FUNCTION_BLOCK FB_MotorWrapper IMPLEMENTS IF_Actuator
VAR_INPUT
END_VAR
VAR_OUTPUT
END_VAR
VAR_IN_OUT
	Axis : AXIS_REF;
END_VAR

VAR
	// MC2 Motion Function Blocks
    fbPower       : MC_Power;
    fbReset       : MC_Reset;
	fbReadStatus  : MC_ReadStatus;
    fbMoveAbs     : MC_MoveAbsolute;
    fbMoveRel     : MC_MoveRelative;
	fbMoveVel	  : MC_MoveVelocity;
	fbSetPos	  : MC_SetPosition;
    fbHome        : MC_Home;
	fbReadPos	  : MC_ReadActualPosition;
    fbStop        : MC_Stop;
	fbHalt		  : MC_Halt;
	fbJog		  : MC_Jog;
    rTrigStop     : R_TRIG;

    fSetPosAbs    : LREAL;
    fSetPosRel    : LREAL;
    bAbsRequest   : BOOL;
    bRelRequest   : BOOL;
    bPowerRequest : BOOL;
    bResetRequest : BOOL;
    bDisableReq   : BOOL;
	
	//Stop()
    bStopExecute     : BOOL;
    bStopRequested   : BOOL;
	bStopDone		 : BOOL;
	
	//GetStatus()
    stStatus       	 : ST_ActuatorStatus;
	stReadStatus	 : ST_AxisReadStatus;
	lastPosition 	 : LREAL := 0.0;
	deltaPos 		 : LREAL;
    bDetectedMovement: BOOL  := FALSE;
    debugSensorValue : BOOL;
	
	//Home()
	bStartDelay		 : BOOL := FALSE;
	tonHoming 		 : TON;
	bhomeExecute	 : BOOL := FALSE;
	bHomeRequest 	 : BOOL := FALSE;

	bExecuteMove	 : BOOL;
	bHomeSensorValue : BOOL;
	bHomeInProgress  : BOOL := FALSE;
	bStartMoveVel	 : BOOL;
	bWaitingForSensorOff : BOOL;
	bWaitingForStop	: BOOL;
	bStartHoming	: BOOL;
	
	//ReadStatus()
	bReadStatusExecute 	: BOOL;
    bReadStatusRequested: BOOL;
	
	//MoveAbs()
	bMoveAbsExecute 	: BOOL;
    bMoveAbsRequested 	: BOOL;
	bMoveAbsDone		: BOOL;
	bMoveAbsStarted		: BOOL;
	rtMoveAbsDone 		: R_TRIG; 
    tonMoveAbs    		: TON;    
    tMoveAbsTout  		: TIME := T#60S;
	tonAbsInWin         : TON;         // estabilidade da janela de posição
	rAbsPosTol          : LREAL := 0.001; // tolerância (ajuste ao teu unit)
	tAbsStable          : TIME  := T#100MS; // estabilidade da janela
	tonAbsTimeout       : TON;         // timeout opcional
	tAbsTimeout         : TIME  := T#60S;   // ajuste conforme curso do eixo
	fbReadVel        	: MC_ReadActualVelocity; // se ainda não existir no FB
	tonVelStill      	: TON;                   // estabilidade de "velocidade ~ 0"
	vTolStill        	: LREAL := 0.0001;       // tolerância de velocidade
	rVelAbs          	: LREAL;                 // auxiliar
	rActPrev         	: LREAL;                 // opcional, se preferir medir Δpos
	
	
	//MoveRel()
	bMoveRelExecute 	: BOOL;
    bMoveRelRequested 	: BOOL;
	bMoveRelDone		: BOOL;
	
	//MoveValve()
	rTargetAngle		: LREAL;
	bMoveValveExecute 	: BOOL;
    bMoveValveRequested : BOOL;
	
	//MoveVel()
	bMoveVelExecute 	: BOOL;
    bMoveVelRequested 	: BOOL;
	bMoveVelDone		: BOOL;
	
	//Reset()
	bResetExecute 		: BOOL;
    bResetRequested 	: BOOL;
	bResetDone			: BOOL;
	
	//SetPosition()
	bSetPosExecute 		: BOOL;
    bSetPosRequested	: BOOL;
	bSetPosDone			: BOOL;
	
	
END_VAR

METHOD Disable : BOOL
VAR_INPUT
END_VAR
// Disable (Remove power from axis)
fbPower(Axis := Axis, Enable := FALSE);
stStatus.bEnabled := FALSE;
stStatus.eState := E_ActuatorState.eDisabled;
Disable := TRUE;
END_METHOD

METHOD Enable : BOOL
VAR_INPUT
END_VAR
// Call MC_Power to enable axis
fbPower(Axis := Axis, Enable := TRUE, Enable_Positive := TRUE, Enable_Negative := TRUE);
stStatus.bEnabled := fbPower.Status;
stStatus.bError := fbPower.Error;
stStatus.iErrorCode := fbPower.ErrorID;
IF fbPower.Error THEN
	stStatus.eState := E_ActuatorState.eError;
	stStatus.sMessage := 'Error in PowerUp';
ELSE
	stStatus.eState := E_ActuatorState.eActive;
END_IF;

Enable := fbPower.Status;
END_METHOD

METHOD GetPosition : LREAL
VAR_INPUT
END_VAR
//Get Actual Position of the motor
//fbReadPos(Axis := Axis, Enable := TRUE);
GetPosition := Axis.NcToPlc.ActPos;
END_METHOD

METHOD GetStatus : ST_ActuatorStatus
VAR_INPUT
END_VAR
// Get unified status struct with all feedback for HMI/diagnostics
fbReadPos(Axis := Axis, Enable := TRUE);
stStatus.fPosition := fbReadPos.Position;
stStatus.bBusy := fbMoveAbs.Busy OR fbMoveRel.Busy OR fbHome.Busy OR fbMoveVel.Busy OR bDetectedMovement;
stStatus.bDone := fbMoveAbs.Done OR fbMoveRel.Done OR fbHome.Done;
stStatus.bError := Axis.Status.Error;

// Calc the position diference
deltaPos := fbReadPos.Position - lastPosition;

IF ABS(deltaPos) > 0.1 THEN
    // Detects forward movement
    IF deltaPos > 0 THEN
		stStatus.bMovingFwd := TRUE;
		stStatus.bMovingBck := FALSE;
		bDetectedMovement   := TRUE;
    // Detects backward movement
    ELSIF deltaPos < 0 THEN
        stStatus.bMovingFwd := FALSE;
        stStatus.bMovingBck := TRUE;
		bDetectedMovement   := TRUE;
    END_IF
ELSE
    // No movement
    stStatus.bMovingFwd := FALSE;
    stStatus.bMovingBck := FALSE;
	bDetectedMovement   := FALSE;
END_IF

lastPosition := fbReadPos.Position;

// Prioritize error messages by source
IF stStatus.bError THEN
	stStatus.eState := E_ActuatorState.eError;
	IF fbPower.Error THEN
		stStatus.sMessage := 'Error in PowerUp';
	ELSIF fbMoveAbs.Error THEN
		stStatus.sMessage := 'Error in MoveAbsolute';
	ELSIF fbMoveRel.Error THEN
		stStatus.sMessage := 'Error in MoveRelative';
	ELSIF fbMoveVel.Error THEN
		stStatus.sMessage := 'Error in MoveVelocity';
	ELSIF fbHome.Error THEN
		stStatus.sMessage := 'Error in Home';
	END_IF
END_IF;

//return
GetStatus := stStatus;
END_METHOD

METHOD Home : BOOL
VAR_INPUT
	pHomeSensor : POINTER TO BOOL; // home sensor pointer
	rVelocity : LREAL;
    rAcc      : LREAL;
    rDec      : LREAL;
	
END_VAR
VAR
	 rTrigHome : R_TRIG;
	 rTrigMove : R_TRIG;
	 rTrigStop : R_TRIG;
END_VAR
bHomeSensorValue  := pHomeSensor^;
IF NOT bHomeRequest THEN
	Home := FALSE;
	bHomeRequest := TRUE;
END_IF

//IF NOT GVL_Motion.bInitialHomingDone THEN
	
	IF bHomeRequest AND NOT bHomeInProgress AND bHomeSensorValue THEN
		bExecuteMove 	:= TRUE;
		bHomeInProgress := TRUE;
	END_IF
	
	IF bHomeRequest AND NOT bHomeInProgress THEN
		bExecuteMove 	:= FALSE;
	
		// If the sensor is already active, skip movement and go to homing directly
		IF NOT bHomeSensorValue THEN
			bStartDelay := TRUE;
			bHomeInProgress := TRUE;
		ELSE
			bExecuteMove := TRUE;
			bHomeInProgress := TRUE;
		END_IF
	END_IF
	
	fbMoveVel(Axis := Axis, Execute := bExecuteMove, Velocity := rVelocity, Acceleration := rAcc, Deceleration := rDec, direction := 1); 
	
	fbStop(Axis := Axis, Execute := bStopExecute, Deceleration := 100);
	
	IF bHomeSensorValue THEN
		//fbMoveVel(Axis := Axis, Execute := bExecuteMove, Velocity := rVelocity, Acceleration := rAcc, Deceleration := rDec, direction := 1); //15, 20, 20
		stStatus.sMessage := 'Seeking home sensor...';
		bStopExecute := FALSE;
	ELSIF NOT bStartDelay THEN
		bExecuteMove := FALSE;
		bStopExecute := TRUE;
		//fbStop(Axis := Axis, Execute := bStopExecute, Deceleration := 10);
	END_IF
	
	IF fbStop.Done THEN
		bStopExecute := FALSE;
		bStartDelay := TRUE;
	END_IF
	
	IF NOT fbStop.Busy THEN
		tonHoming(IN := bStartDelay, PT := T#2S);
	END_IF
	
	IF tonHoming.Q THEN
		bhomeExecute := TRUE;
		stStatus.sMessage := 'Executing MC_Home...';
	END_IF
	
	fbHome(Axis := Axis, Execute := bhomeExecute, Position := 0.0, HomingMode := MC_Direct);
	
	IF fbHome.Done THEN
		stStatus.eState := E_ActuatorState.eIdle;
		stStatus.bError := FALSE;
		stStatus.bDone := TRUE;
		stStatus.sMessage := 'Homing completed';
		bStartDelay  := FALSE;
		bhomeExecute := FALSE;
		tonHoming.IN := FALSE;
		bHomeInProgress := FALSE;
		//GVL_Motion.bMotorsHomeDone := TRUE;
		bHomeRequest := FALSE;
		Home := TRUE;
		RETURN;
	ELSIF fbHome.Error THEN
		stStatus.eState := E_ActuatorState.eError;
		stStatus.bError := TRUE;
		stStatus.iErrorCode := fbHome.ErrorID;
		stStatus.sMessage := 'Error in Homing';
		bhomeExecute := FALSE;
		bStartDelay  := FALSE;
		tonHoming.IN := FALSE;
		bHomeInProgress := FALSE;
		bHomeRequest := FALSE;
		Home := FALSE;
	ELSE
		Home := FALSE;
	END_IF
(*ELSE
	
	IF fbMoveAbs.Done THEN 
		bHomeinProgress := FALSE;
		Home := TRUE;
	END_IF
	
	rTrigMove(CLK := bHomeRequest AND NOT bHomeInProgress);
	
	// If homing previously done then Move to zero position
	fbMoveAbs(Axis := Axis, Execute := rTrigMove.Q, Position := 0, velocity := 15, Acceleration := 15, Deceleration := 15);
	bHomeinProgress := TRUE;
	

	
END_IF*)
END_METHOD

METHOD Jog : BOOL
VAR_INPUT
	bFwd : BOOL;
	bBwd : BOOL;
	//rVelocity : LREAL;
END_VAR
// Call the internal motion block
fbJog(
    Axis := Axis,
    JogForward := bFwd,
    JogBackwards := bBwd,
    Mode := MC_JOGMODE_STANDARD_FAST,
);

// Update actuator status
stStatus.bBusy := fbJog.Busy;
stStatus.bDone := fbJog.Done;
stStatus.bError := fbJog.Error;
stStatus.iErrorCode := fbJog.ErrorID;

Jog := fbJog.Busy;
END_METHOD

METHOD MoveAbsolute : BOOL
VAR_INPUT
	rPosition : LREAL;
    rVelocity : LREAL := 10.0;
    rAcc      : LREAL := 20.0;
    rDec      : LREAL := 20.0;
END_VAR
VAR
	rAct : LREAL;
    rErr : LREAL;
    bInWin : BOOL;
    bStandStill : BOOL;
	opts : ST_MoveOptions;
END_VAR
//Standard Output
MoveAbsolute := FALSE;

// Trigger the command request
IF NOT bMoveAbsRequested THEN
    bMoveAbsExecute := TRUE;
    bMoveAbsRequested := TRUE;
END_IF

// MC_MoveAbsolute function block call
opts.IgnorePositionMonitoring := TRUE;   // Standard practice for move commands

fbMoveAbs(
    Axis := Axis,
    Position := rPosition,
    Execute := bMoveAbsExecute, // Execute flag is controlled by the logic below
    Velocity := rVelocity,
    Acceleration := rAcc,
    Deceleration := rDec,
	options := opts
);

// Release the Execute signal once the block gets in busy or error mode
IF fbMoveAbs.Busy OR fbMoveAbs.Error OR fbMoveAbs.CommandAborted THEN
    bMoveAbsExecute := FALSE;
END_IF

// Flag that movement has successfully started
IF fbMoveAbs.Busy THEN
    bMoveAbsStarted := TRUE;
END_IF

// Status mapping to the wrapper's public status structure
stStatus.bBusy := fbMoveAbs.Busy;
stStatus.bDone := fbMoveAbs.Done;
stStatus.bError := fbMoveAbs.Error;
stStatus.iErrorCode := fbMoveAbs.ErrorID;

//Check if there was any erros on the fbMoveAbs block and resets the trigger
IF bMoveAbsRequested AND bMoveAbsStarted AND 
   	NOT fbMoveAbs.Busy AND NOT fbMoveAbs.Done AND NOT fbMoveAbs.Error THEN
		bMoveAbsRequested := FALSE;
    	bMoveAbsStarted := FALSE;
	
		stStatus.bError := TRUE;
		stStatus.iErrorCode := 9001; // Custom code for 'Motion Aborted/Stuck'
		stStatus.sMessage := 'Movement started but was silently aborted (check external Stop/Power).';
END_IF
	
// Finalization — true Done confirmation
IF bMoveAbsRequested AND fbMoveAbs.Done AND bMoveAbsStarted THEN
    bMoveAbsRequested := FALSE;
	bMoveAbsStarted := FALSE;
    MoveAbsolute := TRUE;
    RETURN;
END_IF

// Abort/error handling
IF fbMoveAbs.CommandAborted THEN
    stStatus.eState := E_ActuatorState.eError;
    stStatus.sMessage := 'Command aborted';
END_IF
IF fbMoveAbs.Error THEN
    stStatus.eState := E_ActuatorState.eError;
    stStatus.sMessage := 'Error in Move Motor';
END_IF
END_METHOD

METHOD MoveRelative : BOOL
VAR_INPUT
	Distance : LREAL;
    Velocity : LREAL := 10.0;
    Acc      : LREAL := 20.0;
    Dec      : LREAL := 20.0;
END_VAR
VAR
END_VAR
// Reuse the same logic from MoveAbsolute
IF NOT bMoveRelRequested THEN
    bMoveRelExecute := TRUE;
    bMoveRelRequested := TRUE;
END_IF

IF fbMoveRel.Busy THEN
    bMoveRelExecute := FALSE;
END_IF

// Call the internal motion block
fbMoveRel(
    Axis := Axis,
    Distance := Distance,
    Execute := bMoveRelExecute,
    Velocity := Velocity,
    Acceleration := Acc,
    Deceleration := Dec
);

// Update actuator status
stStatus.bBusy := fbMoveRel.Busy;
stStatus.bDone := fbMoveRel.Done;
stStatus.bError := fbMoveRel.Error;
stStatus.iErrorCode := fbMoveRel.ErrorID;

IF fbMoveRel.Error THEN
    stStatus.eState := E_ActuatorState.eError;
    stStatus.sMessage := 'Error in Move Motor';
END_IF

IF bMoveRelRequested AND NOT fbMoveRel.Busy AND NOT fbMoveRel.Error THEN
    bMoveRelRequested := FALSE;
    MoveRelative := TRUE;
    RETURN;
ELSE
    MoveRelative := FALSE;
END_IF
END_METHOD

METHOD MoveValve : BOOL
VAR_INPUT
	iPosition : USINT;
	rVelocity : LREAL;
	rAcc	  : LREAL;
	rDec	  : LREAL;
END_VAR
// Map logical valve position to angular position
CASE iPosition OF
    1: rTargetAngle := 0.0;
    2: rTargetAngle := 1200.0;
    3: rTargetAngle := 2400.0;
    4: rTargetAngle := 3600.0;
    5: rTargetAngle := 4800.0;
    6: rTargetAngle := 6000.0;
ELSE
    rTargetAngle := 0;
END_CASE

// Reuse the same logic from MoveAbsolute
IF NOT bMoveValveRequested THEN
    bMoveValveExecute := TRUE;
    bMoveValveRequested := TRUE;
END_IF


// Call the internal motion block
fbMoveAbs(
    Axis := Axis,
    Position := rTargetAngle,
    Execute := bMoveValveExecute,
    Velocity := rVelocity,
    Acceleration := rAcc,
    Deceleration := rDec
);

// Update actuator status
stStatus.bBusy := fbMoveAbs.Busy;
stStatus.bDone := fbMoveAbs.Done;
stStatus.bError := fbMoveAbs.Error;
stStatus.iErrorCode := fbMoveAbs.ErrorID;

IF fbMoveAbs.Busy THEN
    bMoveValveExecute := FALSE;
END_IF

IF fbMoveAbs.Error THEN
    stStatus.eState := E_ActuatorState.eError;
    stStatus.sMessage := 'Error in MoveValve';
END_IF

IF bMoveValveRequested AND NOT fbMoveAbs.Busy AND NOT fbMoveAbs.Error THEN
    bMoveValveRequested := FALSE;
    MoveValve := TRUE;
    RETURN;
ELSE
    MoveValve := FALSE;
END_IF
END_METHOD

METHOD MoveVelocity : BOOL
VAR_INPUT
    rVelocity  : LREAL := 10.0;
    rAcc       : LREAL := 20.0;
    rDec       : LREAL := 20.0;
	iDirection : E_PumpDirection;
END_VAR

VAR
	mcDirection: MC_Direction;
END_VAR
// Reuse the same logic from MoveAbsolute
IF NOT bMoveVelRequested THEN
    bMoveVelExecute := TRUE;
    bMoveVelRequested := TRUE;
END_IF

// Get the corect direction
IF iDirection = E_PumpDirection.Forward THEN
	mcDirection := MC_Direction.MC_Positive_Direction;
	ELSE IF iDirection = E_PumpDirection.Backward THEN
		mcDirection := MC_Direction.MC_Negative_Direction;
	ELSE
		mcDirection := MC_Direction.MC_Current_Direction;
	END_IF
END_IF

// Call the internal motion block
fbMoveVel( 	Axis := Axis,
			Execute := bMoveVelExecute,
			Velocity := rVelocity,
			Direction := mcDirection,
			Acceleration := rAcc,
			Deceleration := rDec
);
			
// Update actuator status
stStatus.bBusy := fbMoveVel.Busy;
stStatus.bError := fbMoveVel.Error;
stStatus.iErrorCode := fbMoveVel.ErrorID;

IF fbMoveVel.Busy THEN
    bMoveVelExecute := FALSE;
END_IF

IF fbMoveVel.Error THEN
    stStatus.eState := E_ActuatorState.eError;
    stStatus.sMessage := 'Error in Move Motor';
END_IF

IF bMoveVelRequested AND NOT fbMoveVel.Busy AND NOT fbMoveVel.Error THEN
    bMoveVelRequested := FALSE;
    MoveVelocity := TRUE;
    RETURN;
ELSE
    MoveVelocity := FALSE;
END_IF
END_METHOD

METHOD ReadStatus : ST_AxisReadStatus
VAR_INPUT
END_VAR
//Method to read status by MC_ReadStatus
Axis.ReadStatus();

//Filling up stReadStatus
stReadStatus.Disabled :=  Axis.Status.Disabled;
stReadStatus.Error := Axis.Status.Error;
stReadStatus.ErrorID := Axis.Status.ErrorID;
stReadStatus.Homed := Axis.Status.Homed;
stReadStatus.Operational := Axis.Status.Operational;
stReadStatus.StandStill := Axis.Status.StandStill;

//Return
ReadStatus := stReadStatus;
END_METHOD

METHOD ReadValveStatus : BOOL
VAR_INPUT
END_VAR
Axis.ReadStatus();

IF Axis.Status.Error AND Axis.Status.ErrorID = 16#00004466 THEN
    ReadValveStatus := FALSE;
ELSE
    ReadValveStatus := NOT Axis.Status.Error AND NOT Axis.Status.Disabled;
END_IF
END_METHOD

METHOD Reset : BOOL
VAR_INPUT
END_VAR
VAR
    (* Local helper to clear flags only on very first call of this reset cycle *)
    bFirstCall : BOOL := FALSE;
	stAxisStat : ST_AxisReadStatus;
END_VAR
// ============================================================================
// 0) Default
// ============================================================================
Reset := FALSE;

// Allways read the actual axis state
Axis.ReadStatus();
stAxisStat.Disabled   			:= Axis.Status.Disabled;
stAxisStat.Error      			:= Axis.Status.Error;
stAxisStat.ErrorID    			:= Axis.Status.ErrorID;
stAxisStat.Homed      			:= Axis.Status.Homed;
stAxisStat.Operational			:= Axis.Status.Operational;
stAxisStat.StandStill 			:= Axis.Status.StandStill;
stAxisStat.MotionCommandsLocked	:= Axis.Status.MotionCommandsLocked;

// 0.1) If the axis is NOT in error, there is nothing to reset.
IF NOT stAxisStat.Error AND NOT stAxisStat.MotionCommandsLocked THEN
    // It guarantees a "clean" status.
    stStatus.bError      := FALSE;
    stStatus.iErrorCode  := 0;
    stStatus.sMessage    := '';
    stStatus.eState      := E_ActuatorState.eIdle;

    // Clear internal reset flags
    bResetRequested      := FALSE;
    bResetExecute        := FALSE;
    bResetDone           := FALSE;

    Reset := TRUE;
    RETURN;
END_IF

// ============================================================================
// 1) Detect new Reset() cycle
// 		- Only enters this section when there is actually an error on the axis
// ============================================================================
IF NOT bResetRequested AND NOT bResetExecute AND NOT bResetDone THEN
    bFirstCall     := TRUE;
    bResetRequested:= TRUE;
END_IF

IF bFirstCall THEN
    // --------------------------------------------------------
    // 1.1) Clears all MC's Executes and internal flags.
    // --------------------------------------------------------
    fbPower(Axis := Axis, Enable := FALSE, Enable_Positive := FALSE, Enable_Negative := FALSE);
    fbMoveAbs(Axis := Axis, Execute := FALSE);
    fbMoveRel(Axis := Axis, Execute := FALSE);
    fbMoveVel(Axis := Axis, Execute := FALSE);
    fbHome(Axis := Axis, Execute := FALSE);
    fbSetPos(Axis := Axis, Execute := FALSE);
    fbStop(Axis := Axis, Execute := FALSE);
    fbHalt(Axis := Axis, Execute := FALSE);
    fbReadStatus(Axis := Axis, Enable := FALSE);
    fbReadPos(Axis := Axis, Enable := FALSE);
	fbReset(Axis := Axis, Execute := FALSE);

    bPowerRequest         := FALSE;
    bDisableReq           := FALSE;

    bAbsRequest           := FALSE;
    bRelRequest           := FALSE;

    bReadStatusRequested  := FALSE;
    bReadStatusExecute    := FALSE;

    // Move Abs
    bMoveAbsRequested     := FALSE;
    bMoveAbsExecute       := FALSE;
    bMoveAbsDone          := FALSE;
    bMoveAbsStarted       := FALSE;

    // Move Rel
    bMoveRelRequested     := FALSE;
    bMoveRelExecute       := FALSE;
    bMoveRelDone          := FALSE;

    // Move Valve
    bMoveValveRequested   := FALSE;
    bMoveValveExecute     := FALSE;

    // Move Vel
    bMoveVelRequested     := FALSE;
    bMoveVelExecute       := FALSE;
    bMoveVelDone          := FALSE;

    // SetPos
    bSetPosRequested      := FALSE;
    bSetPosExecute        := FALSE;
    bSetPosDone           := FALSE;

    // Stop / Halt / Home
    bStopRequested        := FALSE;
    bStopExecute          := FALSE;
    bStopDone             := FALSE;
    bHomeRequest          := FALSE;
    bHomeInProgress       := FALSE;
    bStartHoming          := FALSE;
    bStartMoveVel         := FALSE;
    bWaitingForSensorOff  := FALSE;
    bWaitingForStop       := FALSE;

    // Flags do reset
    bResetRequest         := FALSE;
    bResetRequested       := TRUE;
    bResetDone            := FALSE;

    tonMoveAbs(IN := FALSE);
    tonAbsInWin(IN := FALSE);
    tonHoming(IN := FALSE);
    tonVelStill(IN := FALSE);
    tonAbsTimeout(IN := FALSE);

    rtMoveAbsDone(CLK := FALSE);
    rTrigStop(CLK := FALSE);

    stStatus.bBusy        := FALSE;
    stStatus.bError       := TRUE;             // still error
    stStatus.iErrorCode   := stAxisStat.ErrorID;
    stStatus.sMessage     := 'Resetting axis error...';
    stStatus.eState       := E_ActuatorState.eError;

    bFirstCall := FALSE;
END_IF

// ============================================================================
// 2) Triggers MC_Reset 1x per reset cycle
// ============================================================================
IF bResetRequested AND NOT bResetExecute AND NOT bResetDone THEN
    bResetExecute := TRUE;
END_IF

fbReset(
    Axis    := Axis,
    Execute := bResetExecute
);

// ============================================================================
// 3) MC_Reset error handling
// ============================================================================
IF fbReset.Error THEN
    stStatus.bError      := TRUE;
    stStatus.iErrorCode  := fbReset.ErrorID;
    stStatus.sMessage    := 'Error in MC_Reset';
    stStatus.eState      := E_ActuatorState.eError;

    bResetExecute        := FALSE;
    bResetRequested      := FALSE;
    bResetDone           := FALSE;

    Reset := FALSE;
    RETURN;
END_IF

// MC_Reset's Done
IF fbReset.Done THEN
    bResetExecute := FALSE;
    bResetDone    := TRUE;
END_IF

// ============================================================================
// 4) Finalization: only concludes if the axis really recovered from the error.
// ============================================================================
IF bResetDone AND NOT fbReset.Busy THEN
    // reads the axis status again
    Axis.ReadStatus();
    IF NOT Axis.Status.Error AND NOT Axis.Status.MotionCommandsLocked THEN
        // Success
        stStatus.bError      := FALSE;
        stStatus.iErrorCode  := 0;
        stStatus.sMessage    := '';
        stStatus.eState      := E_ActuatorState.eIdle;

        bResetRequested      := FALSE;
        bResetDone           := FALSE;

        Reset := TRUE;
        RETURN;
    ELSE
        // Still in error (e.g., 0x4650, 0x4260, etc.)
		// Starts another MC_Reset cycle
        bResetDone     := FALSE;
        bResetExecute  := TRUE;
        // Reset remains FALSE until the error is actually cleared.
    END_IF
END_IF


(* Old Reset procedure before 2025's Nov27th
// ============================================================================
// 0) Default return
// ============================================================================
Reset := FALSE;

// ============================================================================
// 1) First call of Reset() in this cycle: clear ALL internal flags and MC executes
// ============================================================================

// If neither a reset request nor a reset execution is active, this is a NEW reset cycle
IF NOT bResetRequested AND NOT bResetExecute AND NOT bResetDone THEN
    bFirstCall := TRUE;
    bResetRequested := TRUE;
END_IF

IF bFirstCall THEN
    // ------------------------------------------------------------
    // 1.1) Clear all MC function block Execute flags
    // ------------------------------------------------------------
    fbPower(Axis := Axis, Enable := FALSE, Enable_Positive := FALSE, Enable_Positive := FALSE);   // Optionally remove power - adapt to your logic
    fbMoveAbs(Axis := Axis, Execute := FALSE);
    fbMoveRel(Axis := Axis, Execute := FALSE);
    fbMoveVel(Axis := Axis, Execute := FALSE);
    fbHome(Axis := Axis, Execute := FALSE);
    fbSetPos(Axis := Axis, Execute := FALSE);
    fbStop(Axis := Axis, Execute := FALSE);
    fbHalt(Axis := Axis, Execute := FALSE);
    fbReadStatus(Axis := Axis, Enable := FALSE);
    fbReadPos(Axis := Axis, Enable := FALSE);

    // ------------------------------------------------------------
    // 1.2) Clear general request / state flags (adapt / extend as needed)
    // ------------------------------------------------------------
    bPowerRequest         := FALSE;
    bDisableReq           := FALSE;

    bAbsRequest           := FALSE;
    bRelRequest           := FALSE;

    bReadStatusRequested  := FALSE;
    bReadStatusExecute    := FALSE;

    // Move Absolute
    bMoveAbsRequested     := FALSE;
    bMoveAbsExecute       := FALSE;
    bMoveAbsDone          := FALSE;
    bMoveAbsStarted       := FALSE;

    // Move Relative
    bMoveRelRequested     := FALSE;
    bMoveRelExecute       := FALSE;
    bMoveRelDone          := FALSE;

    // Move Valve / indexing moves
    bMoveValveRequested   := FALSE;
    bMoveValveExecute     := FALSE;

    // Move Velocity
    bMoveVelRequested     := FALSE;
    bMoveVelExecute       := FALSE;
    bMoveVelDone          := FALSE;

    // Set Position
    bSetPosRequested      := FALSE;
    bSetPosExecute        := FALSE;
    bSetPosDone           := FALSE;

    // Stop / Halt / Jog
    bStopRequested        := FALSE;
    bStopExecute          := FALSE;
    bStopDone             := FALSE;

    // Home-related flags
    bStartHoming          := FALSE;
    bHomeInProgress       := FALSE;
    bHomeRequest          := FALSE;
    bStartMoveVel         := FALSE;
    bWaitingForSensorOff  := FALSE;
    bWaitingForStop       := FALSE;

    // Reset request flags themselves
    bResetRequest         := FALSE;   // if you use this one
    bResetRequested       := TRUE;    // mark that we are inside a reset cycle
    bResetDone            := FALSE;

    // ------------------------------------------------------------
    // 1.3) Clear timers / edge detectors (only inputs; they reset themselves)
    // ------------------------------------------------------------
    tonMoveAbs(IN := FALSE);
    tonAbsInWin(IN := FALSE);
    tonHoming(IN := FALSE);
    tonVelStill(IN := FALSE);
	tonAbsTimeout(IN := FALSE);       

	rtMoveAbsDone(CLK := FALSE);
    rTrigStop(CLK := FALSE);

    // ------------------------------------------------------------
    // 1.4) Clear public status structure
    // ------------------------------------------------------------
    stStatus.bBusy        := FALSE;
    stStatus.bError       := FALSE;
    stStatus.iErrorCode   := 0;
    stStatus.sMessage     := '';
    stStatus.eState       := E_ActuatorState.eIdle; // Back to idle after a successful reset

    // First call handled
    bFirstCall := FALSE;
END_IF

// ============================================================================
// 2) Trigger MC_Reset once per reset cycle
// ============================================================================

// If we still did not start fbReset in this cycle, raise Execute edge
IF bResetRequested AND NOT bResetExecute AND NOT bResetDone THEN
    bResetExecute := TRUE;
END_IF;

// Call MC_Reset
fbReset(
    Axis    := Axis,
    Execute := bResetExecute
);

// ============================================================================
// 3) Handle fbReset state: Busy / Done / Error
// ============================================================================

// 3.1) Error handling
IF fbReset.Error THEN
    stStatus.bError       := TRUE;
    stStatus.iErrorCode   := fbReset.ErrorID;
    stStatus.sMessage     := 'Error in MC_Reset';
    stStatus.eState       := E_ActuatorState.eError;

    // Cancel reset cycle on error
    bResetExecute         := FALSE;
    bResetRequested       := FALSE;
    bResetDone            := FALSE;

    // Return FALSE (reset failed)
    Reset := FALSE;
    RETURN;
END_IF

// 3.2) Normal completion
IF fbReset.Done THEN
    // Drop Execute after Done
    bResetExecute := FALSE;
    bResetDone    := TRUE;
END_IF

// ============================================================================
// 4) Finalization and single-pulse TRUE on function return
// ============================================================================

// When reset is marked as done and fbReset is no longer busy, close the cycle
IF bResetDone AND NOT fbReset.Busy THEN
    // Clear internal reset state for next time
    bResetRequested   := FALSE;
    bResetDone        := FALSE;

    // Optionally ensure axis is not in error and not moving here (if needed)

    // Return TRUE exactly once to the caller
    Reset := TRUE;
	RETURN;
END_IF
*)

(* Old Reset procedure before 2025's Nov24th
// =================================================================================================
// 1) Clear all MC_* Execute flags
// =================================================================================================
fbMoveAbs.Execute := FALSE;
fbMoveRel.Execute := FALSE;
fbMoveVel.Execute := FALSE;
fbHome.Execute    := FALSE;
fbStop.Execute    := FALSE;

// =================================================================================================
// 2) Clear internal request/control flags
// =================================================================================================
bMoveAbsRequested := FALSE;
bMoveRelRequested := FALSE;
bMoveVelRequested := FALSE;
bHomeRequest      := FALSE;

bMoveAbsExecute := FALSE;
bMoveRelExecute := FALSE;
bMoveVelExecute := FALSE;
bHomeExecute    := FALSE;
bStopExecute    := FALSE;

bStopRequested  := FALSE;
bStopDone       := FALSE;

// =================================================================================================
// 3) Reset exposed status (optional, for clean diagnostics after reset)
// =================================================================================================
stStatus.bBusy      := FALSE;
stStatus.bError     := FALSE;
stStatus.iErrorCode := 0;
stStatus.sMessage   := '';
// stStatus.eState  := E_ActuatorState.eIdle;  // keep or set later when success

// =================================================================================================
// 4) Build a clean one-scan pulse for MC_Reset via parameter call
// =================================================================================================

// Generates the pulse just once when it's called
IF NOT bResetRequested THEN
    bResetExecute := TRUE;
    bResetRequested := TRUE;
END_IF

// Reset errors on the axis and motion FBs
IF bResetRequested THEN
    fbReset(Axis := Axis, Execute := bResetExecute);

    stStatus.bError := fbReset.Error;
    stStatus.iErrorCode := fbReset.ErrorID;

    IF fbReset.Error THEN
        stStatus.eState := E_ActuatorState.eError;
        stStatus.sMessage := 'Error in Reset';
        Reset := FALSE;
    ELSE
        stStatus.bError := FALSE;
        stStatus.iErrorCode := 0;
        stStatus.eState := E_ActuatorState.eIdle;
        stStatus.sMessage := '';
    END_IF;
	
	IF bResetDone THEN
        // Flags clearing  
        bResetRequested := FALSE;
        bResetDone := FALSE;
        Reset := TRUE;
        RETURN;
    END_IF
	
    IF fbReset.Done THEN
        bResetExecute := FALSE;
        bResetDone := TRUE;
    END_IF
    
END_IF

// Default Return
Reset := FALSE;
*)
END_METHOD

METHOD SetPosition : BOOL
VAR_INPUT
	rPosition : LREAL;
END_VAR
// Reuse the same logic from MoveAbsolute
IF NOT bSetPosRequested THEN
    bSetPosExecute := TRUE;
    bSetPosRequested := TRUE;
END_IF

// Call the internal motion block
fbSetPos(Axis := Axis, Execute := bSetPosExecute, Position := rPosition, Mode := FALSE);

// Update actuator status
stStatus.bBusy := fbSetPos.Busy;
stStatus.bDone := fbSetPos.Done;
stStatus.bError := fbSetPos.Error;
stStatus.iErrorCode := fbSetPos.ErrorID;

IF fbSetPos.busy THEN
    bSetPosExecute := FALSE;
END_IF

IF fbSetPos.Error THEN
    stStatus.eState := E_ActuatorState.eError;
    stStatus.sMessage := 'Error in motor Set Position';
END_IF

IF bSetPosRequested AND NOT fbSetPos.Busy AND NOT fbSetPos.Error THEN
    bSetPosRequested := FALSE;
    SetPosition := TRUE;
    RETURN;
ELSE
    SetPosition := FALSE;
END_IF
(*
// Call the internal motion block
fbSetPos(Axis := Axis, Execute := bSetPosExecute, Position := rPosition, Mode := FALSE);
*)
END_METHOD

METHOD Stop : BOOL
VAR_INPUT
END_VAR
VAR
END_VAR
// Default output value
Stop := FALSE;

// ============================================================================
// 1) First Stop trigger: set the request flag and generate the rising edge
//    on Execute for MC_Stop
// ============================================================================
IF NOT bStopRequested THEN
    bStopExecute  := TRUE;   // rising edge on MC_Stop.Execute
    bStopRequested := TRUE;
    bStopDone     := FALSE;
END_IF

// ============================================================================
// 2) Safety-net: if Stop was requested but the MC_Stop FB is idle,
//    without Done/Error, and Execute is FALSE (e.g., after a Reset),
//    then re-arm Execute to avoid getting stuck.
// ============================================================================
IF bStopRequested
   AND NOT fbStop.Busy
   AND NOT fbStop.Done
   AND NOT fbStop.Error
   AND NOT bStopExecute THEN
    bStopExecute := TRUE;
END_IF

// ============================================================================
// 3) Call the MC_Stop function block
// ============================================================================
fbStop(Axis := Axis, Execute := bStopExecute);

// ============================================================================
// 4) Internal Stop completion logic (Done / Requested)
// ============================================================================
IF fbStop.Done THEN
    bStopExecute := FALSE;      // release Execute after Done
    bStopDone    := TRUE;
END_IF

IF bStopDone AND NOT fbStop.Busy THEN
    bStopRequested := FALSE;    // stop procedure fully completed
END_IF

// ============================================================================
// 5) Error handling
// ============================================================================
stStatus.bError     := fbStop.Error;
stStatus.iErrorCode := fbStop.ErrorID;

IF fbStop.Error THEN
    stStatus.eState   := E_ActuatorState.eError;
    stStatus.sMessage := 'Error in Stop';
    // Stop remains FALSE; caller must handle Reset() afterwards
    RETURN;
END_IF

// ============================================================================
// 6) Successful completion: update status and return TRUE once
// ============================================================================
IF bStopDone AND NOT fbStop.Busy AND NOT bStopRequested THEN
    stStatus.bError     := FALSE;
    stStatus.iErrorCode := 0;
    stStatus.eState     := E_ActuatorState.eIdle;
    stStatus.sMessage   := 'Axis Stopped';

    // Prepare flags for the next Stop command
    bStopDone := FALSE;

    Stop := TRUE;   // Return TRUE for one cycle
    RETURN;
END_IF

// If execution reaches here, the Stop process is still ongoing
Stop := FALSE;


// Before - changed on Nov 20 2025
(* 
IF NOT bStopRequested THEN
	bStopExecute := TRUE;
	bStopRequested := TRUE;
END_IF

IF bStopRequested THEN
	fbStop(Axis := Axis, Execute := bStopExecute);
END_IF

IF bStopDone AND NOT fbStop.Busy THEN
	bStopRequested := FALSE;
END_IF

IF fbStop.Done THEN
	bStopExecute := FALSE;
	bStopDone := TRUE;
END_IF

stStatus.bError := fbStop.Error;
stStatus.iErrorCode := fbStop.ErrorID;

IF fbStop.Error THEN
	stStatus.eState := E_ActuatorState.eError;
	stStatus.sMessage := 'Error in Stop';
	Stop := FALSE;
END_IF

IF bStopDone AND NOT fbStop.Busy AND NOT bStopRequested THEN
	stStatus.bError := FALSE;
	stStatus.iErrorCode := 0;
	stStatus.eState := E_ActuatorState.eIdle;
	stStatus.sMessage := 'Axis Stopped';
	bStopDone := FALSE;
	Stop := TRUE;
	RETURN;
ELSE
	Stop := FALSE;
END_IF
*)
END_METHOD

END_FUNCTION_BLOCK

(* stored: Version 1.1.0.1, ProductVersion 3.1.4024.15
   POU FB_MotorWrapper: Id {e1ed2152-e06a-419a-985a-88258f9f2422}, SpecialFunc None
   Method Disable: Id {1dc75d36-67d4-446b-8c6d-65221bad79c5}
   Method Enable: Id {d67ddf43-bc97-4342-80c6-577e8cfb8a1b}
   Method GetPosition: Id {4edb2a8e-f8bf-4431-b71c-db3c2d022d41}
   Method GetStatus: Id {a9f2bdab-8820-4977-9409-a8793adba31f}
   Method Home: Id {771f97a4-e7d4-481b-b233-9c33c798e61d}
   Method Jog: Id {3fad885f-82d0-4ede-add0-67a44b600103}
   Method MoveAbsolute: Id {3c2d0047-9043-4f3b-b941-8126a4eab227}
   Method MoveRelative: Id {f57948ef-5e1c-4cbd-b496-9bd6108f8456}
   Method MoveValve: Id {0efdf2ac-cd7b-4dd3-893f-1eab65963717}
   Method MoveVelocity: Id {88eea3e3-3d47-49a5-8a94-a24aaca29cb6}
   Method ReadStatus: Id {75b26eb2-c886-42bf-86aa-71bae3e05caa}
   Method ReadValveStatus: Id {42b9d689-2539-4c89-af9c-94ac21a9a691}
   Method Reset: Id {55ea212e-113c-4739-bf54-01562c1314f2}
   Method SetPosition: Id {a529999b-02b0-40ec-9986-934333a30507}
   Method Stop: Id {27336d58-d763-4c6d-b6e1-79be37906c83} *)
